{attribute 'linkalways'} 
{attribute 'no_explicit_call' := 'This FB is a CLASS and must be accessed using methods or properties'}
{attribute 'enable_dynamic_creation'}
FUNCTION_BLOCK Node_F_VN_AdaptiveThreshold EXTENDS VisionNode
VAR
	ipSrcImage : _ITcVnImage;
    ipDestImage : _ITcVnImage;
    fMaxValue : _LREAL(0.0);
    hrPrev : _HRESULT(S_OK);
	hresult : _HRESULT(S_OK);
END_VAR

METHOD PUBLIC  Clone : I_Node
VAR
	pNode : POINTER TO Node_F_VN_AdaptiveThreshold;
END_VAR
pNode := __NEW(Node_F_VN_AdaptiveThreshold);
Clone := pNode^;
END_METHOD

METHOD FB_init : BOOL
VAR_INPUT
	bInitRetains : BOOL; // if TRUE, the retain variables are initialized (warm start / cold start)
	bInCopyCode : BOOL;  // if TRUE, the instance afterwards gets moved into the copy code (online change)
END_VAR
AddInput('ipSrcImage', ipSrcImage);
AddParameter('fMaxValue', fMaxValue);
AddInput('hrPrev', hrPrev);
AddOutput('ipDestImage', ipDestImage);
AddOutput('hresult', hresult);
END_METHOD

METHOD PROTECTED OnExecute
hresult.Value := F_VN_AdaptiveThreshold(
	ipSrcImage := ipSrcImage.Value,
	ipDestImage := ipDestImage.Value,
    fMaxValue := fMaxValue.Value,
	hrPrev := hrPrev.Value);
END_METHOD

METHOD PUBLIC PreExecutionCheck
VAR_INPUT
	Check : I_PreExecutionChecks;
END_VAR
Check.IsTrue(ipSrcImage.IsValid, 'ipSrcImage must contain an image');
Check.IsTrue(ipSrcImage.HasChannelCount(1), 'ipSrcImage must have 1 channel');
Check.IsTrue(ipSrcImage.IsPixelDepth(8), 'ipSrcImage must have 8 bit pixel depth');
Check.IsTrue((fMaxValue.Value >= 0.0), 'fMaxValue must be greater than or equal to 0');
Check.IsTrue((fMaxValue.Value <= 255.0), 'fMaxValue must be less than or equal to 255');
END_METHOD

END_FUNCTION_BLOCK

(* stored: Version 1.1.0.1, ProductVersion 3.1.4024.15
   POU Node_F_VN_AdaptiveThreshold: Id {681b77bb-ebf8-0d2d-171d-284739fa9ed5}, SpecialFunc None
   Folder Constructor: Id {584e2ced-1903-0042-39c5-84231940ef22}
   Method Clone: Id {c7889fbe-f865-0526-23d7-d12bb9620592}
   Method FB_init: Id {b559bd97-9e3c-001c-212a-3442757e255e}
   Method OnExecute: Id {f4e010b5-106e-09f3-032f-91764639e489}
   Method PreExecutionCheck: Id {04af4b8b-631d-0a7a-0ede-82d17734d041} *)
